PROGRAM MAIN
VAR
	// Blocos MC2
	HabilitaEixo1: MC_Power;
	MoveAbsoluteEixo1: MC_MoveAbsolute;
	MoveRelativeEixo1: MC_MoveRelative;
	HaltEixo1: MC_Halt;
	StopEixo1: MC_Stop;
	// Variáveis de controle e auxílio
	bHabilitaEixo1: BOOL;
	bMoverAbsoluto: BOOL;
	bMoverRelativo: BOOL;
	bParadaSuave: BOOL;
	bParadaTravada: BOOL;
	bComandoConcluido: BOOL;
	uEstadoEixo : UDINT;
END_VAR

//Ler status
Eixos.Eixo1.ReadStatus()
;
// Mostra o Estado do Eixo 1
uEstadoEixo := Eixos.Eixo1.NcToPlc.AxisState
;
// Indica se houve Done por parte de algum dos blocos
IF MoveAbsoluteEixo1.Done OR MoveRelativeEixo1.Done THEN
	bComandoConcluido := TRUE;
END_IF

//Habilitar Eixo 1
HabilitaEixo1(
	Axis:= Eixos.Eixo1, 
	Enable:= bHabilitaEixo1, 
	Enable_Positive:= bHabilitaEixo1, 
	Enable_Negative:= bHabilitaEixo1, 
	Override:= 100)
;
// Move Absolute Eixo 1
MoveAbsoluteEixo1(
	Axis:= Eixos.Eixo1, 
	Execute:= bMoverAbsoluto, 
	Position:= 50, 
	Velocity:= 50)
;
// Move Relative Eixo 1
MoveRelativeEixo1(
	Axis:= Eixos.Eixo1, 
	Execute:= bMoverRelativo, 
	Distance:= 20, 
	Velocity:= 20)
;
// Parar o Eixo 1
HaltEixo1(
	Axis:= Eixos.Eixo1, 
	Execute:= bParadaSuave)
;
// Parar o Eixo 1 e impedir que se mova até que  desative o bloco Stop
StopEixo1(
	Axis:= Eixos.Eixo1, 
	Execute:= bParadaTravada)
;

END_PROGRAM

(* stored: Version 1.1.0.1
   POU MAIN: Id {3bf0370f-8f08-460a-b5b6-c7e00346ad17}, SpecialFunc None *)
